Universal Robots PolyScope program: 07_Force_measurement_01.urp

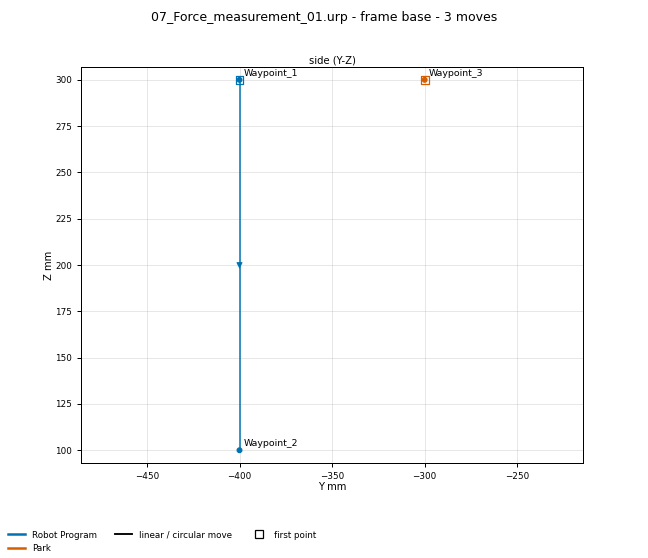
[picture p0: tool path of 07_Force_measurement_01.urp in frame base, 3 of 3 moves have a stored position in this frame; points joined in program order, loops and branches not executed]
Program 07_Force_measurement_01 (installation=default directory=/home/ur/ursim-current/programs/Test_Programs createdIn=5.9.1.1031110 lastSavedIn=5.9.1.1031110 robotSerialNumber=20195599999)
Calibrated DH parameters: a=[0, -0.425, -0.3922, 0, 0, 0]; d=[0.1625, 0, 0, 0.1333, 0.0997, 0.0996]; alpha=[1.570796, 0, 0, 1.570796, -1.570796, 0]; deltaTheta=[0, 0, 0, 0, 0, 0]
InitVariablesNode
Robot Program (runOnlyOnce=false)
  MoveL speed 250 mm/s, acceleration 1200 mm/s^2 (useActiveTCP=true) feature=Base
    Waypoint Waypoint_1: TCP in base x=0 y=-400 z=300 mm, rx=0 ry=3.1416 rz=0 rad; joints [-70.534, -80.53, -127.136, -62.333, 90, 19.466] deg
  Force Simple feature=Base; selection=[0, 0, 1, 0, 0, 0]; wrench=[0, 0, 10, 0, 0, 0]; limitsForce=[0.15, 0.15, 0.15, 1.047198, 1.047198, 1.047198]; limitsMotion=[0.1, 0.1, 0.1, 0.349066, 0.349066, 0.349066]
    MoveL speed 250 mm/s, acceleration 1200 mm/s^2 (useActiveTCP=true) feature=Base
      Waypoint Waypoint_2: TCP in base x=0 y=-400 z=100 mm, rx=0 ry=3.1416 rz=0 rad; joints [-70.534, -108.612, -140.194, -21.194, 90, 19.466] deg
  If Fmax≟1
    Call Park
SubProgram -> Park
Event  expression=ForceValue>40
  Fmax := 1
  Set DigitalOutput pin=digital_out[0]; digitalValue=1
Thread Thread_1 (runOnlyOnce=false)
  Wait Sleep waitTime=0.01
  ForceValue := force()
SubProgram Park (keepSynchronizedWithDisk=false)
  MoveL speed 250 mm/s, acceleration 1200 mm/s^2 (useActiveTCP=true) feature=Base
    Waypoint Waypoint_3: TCP in base x=0 y=-300 z=300 mm, rx=0 ry=3.1416 rz=0 rad; joints [-63.619, -62.29, -138.492, -69.218, 90, 26.381] deg
    Set DigitalOutput pin=digital_out[0]; digitalValue=0
    Wait Sleep waitTime=3
    Fmax := 0
